# B&R Automation Studio project POMIRS__MukhortovAA_KVBO-07-22
Automation Studio 4.5.2.102

## Configuration Config1

### Task classes (Cpu.sw)
```
Cyclic#1:
  Program <- Program.prg
Binaries: udbdef, TCData, iomap, ashwac, Role, sysconf, arconfig, asfw, User, ashwd
Libraries: MotorContr
```

### Hardware
```
4PP065_0571_P74 : 4PP065.0571-P74 v1.1.2.0
  Connector IF5:
    ActivateDevice = 1
  ConfigurationID = labBR
  Simulation = 1
```

## Logical view

Binary libraries used (declarations not repeated): operator, runtime, astime, AsIecCon

### Library Logical/Libraries/MotorContr (ANSIC)

#### MotorContr.fun - Exported functions and function blocks
```iecst
{REDUND_ERROR} FUNCTION_BLOCK FB_Motor (*TODO: Add your comment here*) (*$GROUP=User,$CAT=User,$GROUPICON=User.png,$CATICON=User.png*)
	VAR_INPUT
		u : REAL;
	END_VAR
	VAR_OUTPUT
		w : REAL;
		phi : REAL;
	END_VAR
	VAR
		speed_integrator : FB_Integrator;
		position_integrator : FB_Integrator;
		Tm : REAL;
		ke : REAL;
		dt : REAL;
	END_VAR
END_FUNCTION_BLOCK

{REDUND_ERROR} FUNCTION_BLOCK FB_Regulator (*TODO: Add your comment here*) (*$GROUP=User,$CAT=User,$GROUPICON=User.png,$CATICON=User.png*)
	VAR_INPUT
		e : REAL;
	END_VAR
	VAR_OUTPUT
		u : REAL;
	END_VAR
	VAR
		k_p : REAL;
		k_i : REAL;
		integrator : FB_Integrator;
		iyOld : REAL;
		max_abs_value : REAL;
		dt : REAL;
		e_p : USINT;
	END_VAR
END_FUNCTION_BLOCK

{REDUND_ERROR} FUNCTION_BLOCK FB_Integrator (*TODO: Add your comment here*) (*$GROUP=User,$CAT=User,$GROUPICON=User.png,$CATICON=User.png*)
	VAR_INPUT
		in : REAL;
	END_VAR
	VAR_OUTPUT
		out : REAL;
	END_VAR
	VAR
		dt : REAL;
	END_VAR
END_FUNCTION_BLOCK
```

#### FB_Motor.c
```c
#include <bur/plctypes.h>
#ifdef __cplusplus
	extern "C"
	{
#endif
	#include "MotorContr.h"
#ifdef __cplusplus
	};
#endif

void FB_Motor(struct FB_Motor* inst)
{
    /*
    REAL a = inst->u / inst->ke - inst->w;
    REAL b = a / inst->Tm;

    inst->integrator.in = b;
    FB_Integrator(&inst->integrator);

    inst->w = inst->integrator.out;

    inst->integrator.in = inst->w * inst->dt;
    FB_Integrator(&inst->integrator);

    inst->phi = inst->integrator.out;
    */

    inst->speed_integrator.in = (inst->u / inst->ke - inst->w) / inst->Tm;;
    inst->speed_integrator.dt = inst->dt;
    FB_Integrator(&inst->speed_integrator);
    inst->w = inst->speed_integrator.out;

    inst->position_integrator.in = inst->w;
    inst->position_integrator.dt = inst->dt;
    FB_Integrator(&inst->position_integrator);
    inst->phi = inst->position_integrator.out;

}
```

#### FB_Regulator.c
```c
#include <bur/plctypes.h>
#ifdef __cplusplus
	extern "C"
	{
#endif
	#include "MotorContr.h"
#ifdef __cplusplus
	};
#endif
/* TODO: Add your comment here */
void FB_Regulator(struct FB_Regulator* inst)
{/*
    REAL a = inst->e * inst->k_p;
    REAL b = inst->e * inst->k_i * inst->dt;

    inst->integrator.in = b + inst->iyOld;
    FB_Integrator(&inst->integrator);
    if (a > inst->max_abs_value || a < -inst->max_abs_value) {
        if (a > 0) a = inst->max_abs_value;
        else a = -inst->max_abs_value;
    }

    a += inst->integrator.out;
    if (a < inst->max_abs_value && a > -inst->max_abs_value)
        inst->u = a;
    else
    {
        if (a > 0) inst->u = inst->max_abs_value;
        else inst ->u = -inst->max_abs_value;
    }

    inst->iyOld = inst->u - a;
*/

    REAL p_term = inst->e * inst->k_p;
    REAL i_term_input = inst->e * inst->k_i * inst->dt;

    i_term_input += inst->iyOld;

    inst->integrator.in = i_term_input;
    FB_Integrator(&inst->integrator);

    REAL unlimited_u = p_term + inst->integrator.out;

    if (unlimited_u > inst->max_abs_value) {
        inst->u = inst->max_abs_value;
    } else if (unlimited_u < inst->max_abs_value) {
        inst->u = -inst->max_abs_value;
    } else {
        inst->u = unlimited_u;
    }

    inst->iyOld = inst->u - unlimited_u;

}
```

#### FB_Integrator.c
```c
#include <bur/plctypes.h>
#ifdef __cplusplus
	extern "C"
	{
#endif
	#include "MotorContr.h"
#ifdef __cplusplus
	};
#endif
/* TODO: Add your comment here */
void FB_Integrator(struct FB_Integrator* inst)
{
    inst->out += inst->in*inst->dt;
}
```

### Program Logical/Program

#### Variables.var
```iecst
VAR
	fb_controller : FB_Regulator;
	fb_motor : FB_Motor;
	fb_motor1 : FB_Motor;
	Speed : REAL;
	Enable : BOOL;
	count : INT;
END_VAR
```

#### Cyclic.c
```c
#include <bur/plctypes.h>
#include <bur/plc.h>

#ifdef _DEFAULT_INCLUDES
	#include <AsDefault.h>
#endif

void _CYCLIC ProgramCyclic(void)
{
    if(Enable)
    {

        count += 1;

        if (count >= 1000 && count <= 1500) Speed = 40;
        else Speed = 5;

        fb_controller.e = Speed - fb_motor.w;

        fb_motor.u = Speed * fb_motor.ke;
        fb_motor1.u = (Speed - fb_controller.u) * fb_motor1.ke;

        FB_Regulator(&fb_controller);
        FB_Motor(&fb_motor);
        FB_Motor(&fb_motor1);

        /*
        count += 1;

        if (count >= 1000 && count <= 1500) Speed = 40;
        else Speed = 5;

        fb_controller.e = Speed - fb_motor.w;

        FB_Regulator(&fb_controller);

        fb_motor.u = fb_controller.u;
        fb_motor1.u = Speed * fb_motor1.ke;

        FB_Motor(&fb_motor);
        FB_Motor(&fb_motor1);   */
    }
    else Speed = 0;
}
```

#### Exit.c
```c
#include <bur/plctypes.h>

#ifdef _DEFAULT_INCLUDES
	#include <AsDefault.h>
#endif

void _EXIT ProgramExit(void)
{

}
```

#### Init.c
```c
#include <bur/plctypes.h>

#ifdef _DEFAULT_INCLUDES
	#include <AsDefault.h>
#endif

void _INIT ProgramInit(void)
{
    count = 0;
    Speed = 0;
    Enable = 1;

    fb_motor.speed_integrator.dt = 0.02;
    fb_motor.speed_integrator.out = 0;

    fb_motor.position_integrator.dt = 0.02;
    fb_motor.position_integrator.out = 0;

    fb_motor.dt = 0.02;
    fb_motor.ke = 43.98;
    fb_motor.Tm = 0.173;

    fb_motor1.speed_integrator.dt = 0.02;
    fb_motor1.speed_integrator.out = 0;

    fb_motor1.position_integrator.dt = 0.02;
    fb_motor1.position_integrator.out = 0;

    fb_motor1.dt = 0.02;
    fb_motor1.ke = 43.98;
    fb_motor1.Tm = 0.173;

    fb_controller.dt = 0.02;
    fb_controller.k_p = 3.804;
    fb_controller.k_i = 21.99;
    fb_controller.max_abs_value = 24;

    //fb_motor.integrator.dt = 0.02;
    //fb_motor1.integrator.dt = 0.02;
    fb_controller.integrator.dt = 0.02;
}
```

Listed in the project but not available here: Logical/Libraries/MotorContr/Types.typ, Logical/Libraries/MotorContr/Constants.var
